(* CoDeSys 2.3 export: FBK16PUMPSCONTROL.EXP *)

(* POU K16/fbK16PumpsControl, ST *)
FUNCTION_BLOCK fbK16PumpsControl
(*
	Управление насосами К16
	контура ГВС
*)
VAR CONSTANT
	PumpCheckDelayTime : TIME := T#2s;
	PumpWorkHeatingOrder : ARRAY [1..MAX_K16_PUMPS_NUM] OF USINT := 1, 2;
END_VAR
VAR_INPUT
	ManualMode: BOOL;						(*Ручной режим?*)
	WorkAllowed: BOOL;					(*Работа разрешена?*)
	EmergencyPumpStopButtonPressed: ARRAY [1..MAX_K16_PUMPS_NUM] OF BOOL; (*Нажат аварийный стоп насоса?*)
	PumpState: ARRAY [1..MAX_K16_PUMPS_NUM] OF BOOL;	(*Работает насос?*)
	PressureDrop : BOOL;					(*Есть разница давлений?*)
END_VAR
VAR_OUTPUT
END_VAR
VAR
	pumpStatusCheckDelay	: ARRAY [1..MAX_K16_PUMPS_NUM] OF TON;
	pumpsTrainingControl : fbK16PumpsTraining;
END_VAR

VAR_TEMP
	i : USINT;
	pumpWorkOrder : ARRAY [1..MAX_K16_PUMPS_NUM] OF USINT;
	pumpStatusCheck : ARRAY [1..MAX_K16_PUMPS_NUM] OF BOOL;
	break : BOOL := FALSE;
END_VAR
FOR i := 1 TO MAX_K16_PUMPS_NUM DO
	pumpStatusCheckDelay[i](IN := PumpState[i], PT := PumpCheckDelayTime);
	pumpStatusCheck[i] := pumpStatusCheckDelay[i].Q;
END_FOR;

fK16PumpsFaultyControl(
	PumpState				:= PumpState,
	PumpStatusCheckDelay	:= pumpStatusCheck,
	PressureDrop			:= PressureDrop
);

IF ManualMode THEN (*Ручной режим?*)
(*
	FOR i := 1 TO MAX_K16_PUMPS_NUM DO
		fK16PumpManualControl(
			PumpID	:= i,
			TurnOn	:= TurnOnPumpButtonPressed[i],
			TurnOff	:= TurnOffPumpButtonPressed[i],
			State		:= PumpState[i],
			EmergencyStop := EmergencyPumpStopButtonPressed[i]
		);
	END_FOR;
*)
	(*Контроллер никак не участвует в ручном режиме*)
	FOR i := 1 TO MAX_K16_PUMPS_NUM DO
		fTurnOffK16Pump(i);
	END_FOR;
ELSE
	IF WorkAllowed THEN	(*Работа разрешена?*)
		pumpWorkOrder := PumpWorkHeatingOrder;
		FOR i := 1 TO MAX_K16_PUMPS_NUM DO
			(*
				работаем с насосами в порядке их приоритета
				Ищем первый исправный насос и включаем его
			*)
			IF NOT(break) AND NOT(K16PumpFaulty[pumpWorkOrder[i]]) THEN
				fK16PumpAutoControl(
						PumpID := pumpWorkOrder[i],
						EmergencyPumpStopButtonPressed := EmergencyPumpStopButtonPressed[pumpWorkOrder[i]]
				);
				break := TRUE;
			END_IF;
		END_FOR;
		(*периодическая тренировка насосов*)
		pumpsTrainingControl();
	ELSE
		(*
			если работа не разрешена,
			выключаем все насосы
		*)
		FOR i := 1 TO MAX_K16_PUMPS_NUM DO
			fTurnOffK16Pump(i);
		END_FOR;
		RETURN;
	END_IF;
END_IF;
END_FUNCTION_BLOCK
